{attribute addProperty BoxType "EJ1914-0000-0017"}
{attribute addProperty Id "FSoE_InputsFSoE_Inputs_899BAC0E486FSoE_OutputsFSoE_Outputs_E28701A0486"}
{attribute addProperty CRC "1620154689"}
{attribute addProperty SizeInBites "96"}
{attribute addProperty SizeInBytes "12"}
TYPE Module_1_FSOE_60919941 :
STRUCT
	{attribute addProperty Name "FSoE_Inputs"}
	FSoE_Inputs  : FSoE_Inputs_899BAC0E;
	{attribute addProperty Name "FSoE_Outputs"}
	FSoE_Outputs  : FSoE_Outputs_E28701A0;
END_STRUCT
END_TYPE

(* stored: Version 1.2.0.0, ProductVersion 3.1.4024.9
   DUT Module_1_FSOE_60919941: Id {eca6a4d5-0463-47e3-994e-9ae7d727240a} *)
